# EPICS substitutions: viocs/ts_ps/ts_psApp/Db/septa.substitutions
file "db/septa.db" {
    pattern { family, pos }
        { "SEPTUMEXT", "01" }
        { "SEPTUMTHICK", "04"}
        { "SEPTUMTHIN", "04"}
}
